(* PLC project real2int_scale, Dassault Systèmes ControlBuild 2024x *)
(* stored: creationDateTime 2023-10-03T11:13:31-01:00 *)

(* This module simulates a scaling of a real into an integer. Form of the scaling equation is y = k x . *)
FUNCTION_BLOCK equipment_library.real2int_scale
  VAR_INPUT
    inputValue : REAL := 0.0;
  END_VAR
  VAR_OUTPUT
    dintValue : DINT := 0;
    intValue : INT := 0;
  END_VAR
  VAR CONSTANT
    coefficient : REAL := 1.0;
    offset : REAL := 0.0;
  END_VAR
  VAR
    d_scale : BOOL := false;
    v_d_scale : DINT := 0;
  END_VAR


ACTION C_source_code:
/* ----------------------------------------------------------------	*/
/* Type : Model of Operative Behaviour					*/
/* Category :  Toolbox							*/
/* Author : Dassault Systemes						*/
/* Update date : June 2018						*/
/* ----------------------------------------------------------------	*/
/* This module simulates a scaling of a real into an integer	 	*/
/*	by multiplying it by a parameter coefficient.			*/
/* Form of the scaling equation is y = k x .				*/
/* ----------------------------------------------------------------	*/

if (d_scale)
	dintValue = v_d_scale;
else
	dintValue = (inputValue * coefficient) + offset;

if ((dintValue >= -32768) && (dintValue <= 32767)) 
	intValue = dintValue ;
else 
	intValue = 0;
END_ACTION
END_FUNCTION_BLOCK
